// TIA Portal V17 export
BLOCK "FC_Move"   // ObjectSW14, LAD
BEGIN

REGION Network 1: move convert mux
END_REGION
END_BLOCK
